Fanuc KAREL source: kt00074.KL

-- PROVISIONAL review KL for V770-1; original PC SHA256 04519cff8470600194c3ee49c998cd28c2b64e7e760b7b24c916afa84ad7272c
-- Incomplete behavior may be omitted. Consult companion uncertainty JSON. Do not deploy.
PROGRAM KT00074
%NOLOCKGROUP
VAR
  R1 : REAL
  I2 : INTEGER
  OUT : REAL
BEGIN
  -- UNRESOLVED_PC offsets 5-16; opcodes 2E,23
  -- UNRESOLVED_PC offsets 21-32; opcodes 2E,23
  -- UNRESOLVED_PC offsets 37-57; opcodes 21,21,64,6B,23
  -- UNRESOLVED_PC offsets 62-66; opcodes 7F
END KT00074
